FUNCTION_BLOCK IA_RHS (* ISOBUS Adapter for Rear Hitch Status (RHS) *)
  (* Standard: ISO 11783-7; Classification: PGN 65093; Description: Copyright (c) 2024-2026 HR Agrartechnik GmbH This program and the accompanying materials are made available under the terms of the Eclipse Public License 2.0 which is available at https://www.eclipse.org/legal/epl-2.0/ SPDX-License-Identifier: EPL-2.0 *)
  (* Version 1.2, 2026-09-17, Franz Höpfinger, HR Agrartechnik GmbH, Bugfix (Franz: 'IA_VDS hat einen Bug, moeglicherweise alle anderen auch'): .IND->TIMEOUT.E1 ergaenzt (analog IA_VDS) - bisher wurde TIMEOUT.E1 NUR von .TIMEOUT gefeuert (Timeout-Beginn), nie beim Eintreffen einer normalen Botschaft (.IND) - TIMEOUT.D1 (Q_timeout=FALSE) wurde also gesetzt, aber nie an den TIMEOUT-Plug propagiert, sobald der Timeout wieder endete. *)
  (* Version 1.1, 2026-09-16, Franz Höpfinger, HR Agrartechnik GmbH, E_D_FF_ANY-Aenderungsfilter fuer POSITION/FORCE/DRAFT ergaenzt (analog IA_RPTO v1.1). *)
  PACKAGE isobus::tecu;
  (* Documentation:
  ISOBUS Adapter for Rear Hitch Status (RHS)
   TIMEOUT.E1-Verdrahtung: I_CORE.TIMEOUT (echter Timeout-Eintritt) UND I_CORE.IND (Normalbetrieb) sind beide auf den Adapter-Plug TIMEOUT.E1 verdrahtet - bewusst so, damit TIMEOUT.D1 (Q_timeout) am Adapter-Plug auch beim Zuruecksetzen auf false aktualisiert wird, nicht nur beim Eintreten des Timeouts. Der zugrundeliegende TIMEOUT/IND-Vertrag von I_CORE selbst ist in dessen eigener .fbt-Datei dokumentiert.
  *)
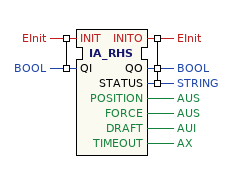
  EVENT_INPUT
    INIT : EInit WITH QI; (* Service Initialization *)
  END_EVENT
  EVENT_OUTPUT
    INITO : EInit WITH QO, STATUS; (* Initialization Confirm *)
  END_EVENT
  VAR_INPUT
    QI : BOOL; (* Event Input Qualifier *)
  END_VAR
  VAR_OUTPUT
    QO : BOOL; (* Event Output Qualifier *)
    STATUS : STRING;
  END_VAR
  PLUGS
    POSITION : adapter::types::unidirectional::AUS; (* Rear Hitch Position *)
    FORCE : adapter::types::unidirectional::AUS; (* Rear Nominal Lower Link Force *)
    DRAFT : adapter::types::unidirectional::AUI; (* Rear Draft *)
    TIMEOUT : adapter::types::unidirectional::AX; (* Timeout Status *)
  END_PLUGS
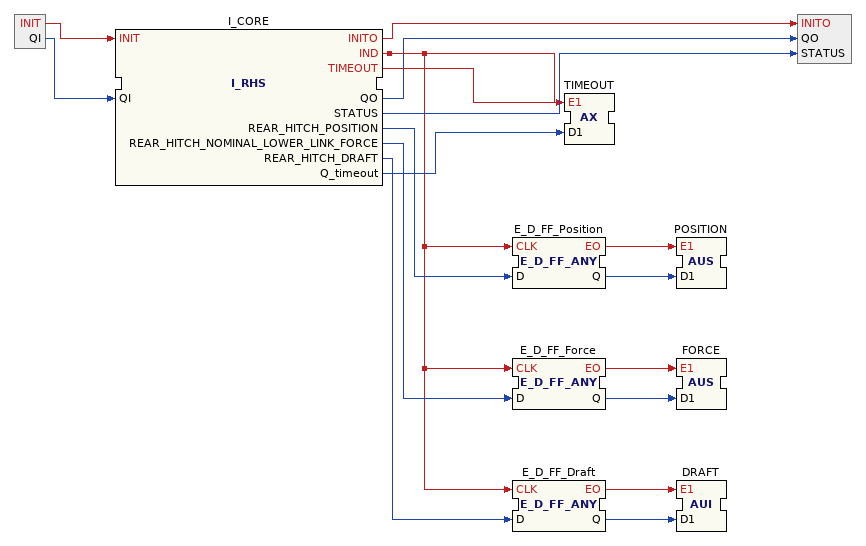
  FBS
    I_CORE : isobus::tecu::I_RHS;
    E_D_FF_Position : iec61499::events::E_D_FF_ANY;
    E_D_FF_Force : iec61499::events::E_D_FF_ANY;
    E_D_FF_Draft : iec61499::events::E_D_FF_ANY;
  END_FBS
  EVENT_CONNECTIONS
    INIT TO I_CORE.INIT;
    I_CORE.INITO TO INITO;
    I_CORE.IND TO E_D_FF_Position.CLK;
    E_D_FF_Position.EO TO POSITION.E1;
    I_CORE.IND TO E_D_FF_Force.CLK;
    E_D_FF_Force.EO TO FORCE.E1;
    I_CORE.IND TO E_D_FF_Draft.CLK;
    E_D_FF_Draft.EO TO DRAFT.E1;
    I_CORE.TIMEOUT TO TIMEOUT.E1;
    I_CORE.IND TO TIMEOUT.E1;
  END_CONNECTIONS
  DATA_CONNECTIONS
    QI TO I_CORE.QI;
    I_CORE.QO TO QO;
    I_CORE.STATUS TO STATUS;
    I_CORE.REAR_HITCH_POSITION TO E_D_FF_Position.D;
    E_D_FF_Position.Q TO POSITION.D1;
    I_CORE.REAR_HITCH_NOMINAL_LOWER_LINK_FORCE TO E_D_FF_Force.D;
    E_D_FF_Force.Q TO FORCE.D1;
    I_CORE.REAR_HITCH_DRAFT TO E_D_FF_Draft.D;
    E_D_FF_Draft.Q TO DRAFT.D1;
    I_CORE.Q_timeout TO TIMEOUT.D1;
  END_CONNECTIONS
END_FUNCTION_BLOCK
